// Mitsubishi GX Works2 project: 05.01Group17Final   PLC: FX3G

// global labels: Global1
VAR_GLOBAL
  Start_Day AT X007 : BOOL;
  Y_7 AT Y007 : BOOL;
  FillZilofKazefet AT X011 : BOOL;
  HelpLight AT M34 : BOOL;
  BlinkingLight AT M4 : BOOL;
  BlinkingTimer1 AT TC0 : BOOL;
  ConstantBlinking AT K5 : INT;
  TimerValue1 AT TS0 : BOOL;
  BlinkingLight2 AT M5 : BOOL;
  BlinkingTimer2 AT TC1 : BOOL;
  TimerValue2 AT TS1 : BOOL;
  BlinkingLightStop AT M5 : BOOL;
  StopBlinking AT TS4 : BOOL;
  Timer4 AT TC4 : BOOL;
  EndDay AT K30 : INT;
  BlinkingLightStop1 AT M6 : BOOL;
  CHOCOLATE AT D1111 : REAL;
  CREAM_STOCK AT D1118 : REAL;
  CHOCOLATE_STOCK AT D1121 : REAL;
  BISCUIT_STOCK AT D1124 : REAL;
END_VAR
VAR_GLOBAL CONSTANT
  C_300 : REAL := 300;
  C_260 : INT := 600;
  C_240 : REAL := 240;
  B_6 : REAL := 6;
END_VAR
VAR_GLOBAL
  VALID AT M2 : BOOL;
  CREAM AT D1100 : REAL;
  BISCUIT AT D1113 : REAL;
  X1_touch AT X001 : BOOL;
  X2_Cam AT X002 : BOOL;
  X5_error AT X005 : BOOL;
  System_on AT M0 : BOOL;
  x3_Sen_30 AT X003 : BOOL;
  X4_sen_15 AT X004 : BOOL;
  Spirk_system AT Y004 : BOOL;
  shut_Down AT X007 : BOOL;
  Start_sys AT X010 : BOOL;
  moveCream AT X011 : BOOL;
  sprinklingContainer AT D1127 : REAL;
END_VAR
VAR_GLOBAL CONSTANT
  nimus_300 : REAL := 300;
  minus_300 : REAL := 300;
  minus_6 : REAL := 6;
END_VAR
VAR_GLOBAL
  M_10 AT M10 : BOOL;
  TimerShinua AT TC10 : BOOL;
END_VAR
VAR_GLOBAL CONSTANT
  shinua : INT := 40;
END_VAR
VAR_GLOBAL
  shinuaFinished AT TS10 : BOOL;
  Y_0 AT Y000 : BOOL;
  Y_1 AT Y001 : BOOL;
  analogCheck AT X006 : BOOL;
  analogInput1 AT D8280 : INT;
  saveAnalog1 AT D1300 : INT;
END_VAR
VAR_GLOBAL CONSTANT
  lessThan : INT := 5;
  lessthan_10 : INT := 10;
  moreThan_6 : INT := 6;
END_VAR
VAR_GLOBAL
  less_10 : BOOL;
  Be0_5 AT M55 : BOOL;
  Be6_10 AT M56 : BOOL;
END_VAR
VAR_GLOBAL CONSTANT
  regularTzipuy : REAL := 120;
  doubleTzipuy : REAL := 240;
END_VAR
VAR_GLOBAL
  dipContainer AT D1132 : REAL;
  TimerDip AT TC8 : BOOL;
END_VAR
VAR_GLOBAL CONSTANT
  timer5 : INT := 50;
END_VAR
VAR_GLOBAL
  TS_8 AT TS8 : BOOL;
  Y_3 AT Y003 : BOOL;
  Gelem AT M80 : BOOL;
END_VAR
VAR_GLOBAL CONSTANT
  div400 : INT := 400;
END_VAR
VAR_GLOBAL
  M_100 AT M100 : BOOL;
  M_101 AT M101 : BOOL;
  ariza AT X000 : BOOL;
  countUnits AT CC0 : BOOL;
END_VAR
VAR_GLOBAL CONSTANT
  Equal_5 : REAL;
END_VAR
VAR_GLOBAL
  Y_2 AT Y002 : BOOL;
END_VAR
VAR_GLOBAL CONSTANT
  Mishtane : INT := 5;
END_VAR
VAR_GLOBAL
  CS_0 AT CS0 : BOOL;
  countUnits2 AT CC1 : BOOL;
END_VAR
VAR_GLOBAL CONSTANT
  until6 : INT := 6;
END_VAR
VAR_GLOBAL
  CS_1 AT CS1 : BOOL;
  rst_ziluf AT M60 : BOOL;
END_VAR
VAR_GLOBAL CONSTANT
  div10 : INT := 10;
END_VAR
VAR_GLOBAL
  Output_Analog1 AT D1150 : INT;
END_VAR
VAR_GLOBAL CONSTANT
  E_120 : INT := 120;
  E_240 : INT := 240;
  plus20 : INT := 20;
  limit : INT := 6;
  add_6 : INT := 6;
END_VAR
VAR_GLOBAL
  closeCount AT M77 : BOOL;
  M_EZER AT M99 : BOOL;
  M_reCheck AT M88 : BOOL;
END_VAR
VAR_GLOBAL CONSTANT
  last_6 : INT := 6;
END_VAR
VAR_GLOBAL
  count_last_6 AT CC12 : BOOL;
  EndOfDay AT CS12 : BOOL;
  analogOutput AT D8282 : INT;
END_VAR
VAR_GLOBAL CONSTANT
  mul40 : INT := 40;
END_VAR

// task Task_01 (event TRUE, interval 0, priority 31): POU_01

PROGRAM POU_01
VAR CONSTANT
  plus_one : INT := 1;
END_VAR
(* structured ladder/FBD written out as ST: instructions are called as NAME(EN, inputs, outputs); _pN, _eN, _tN stand for wires *)
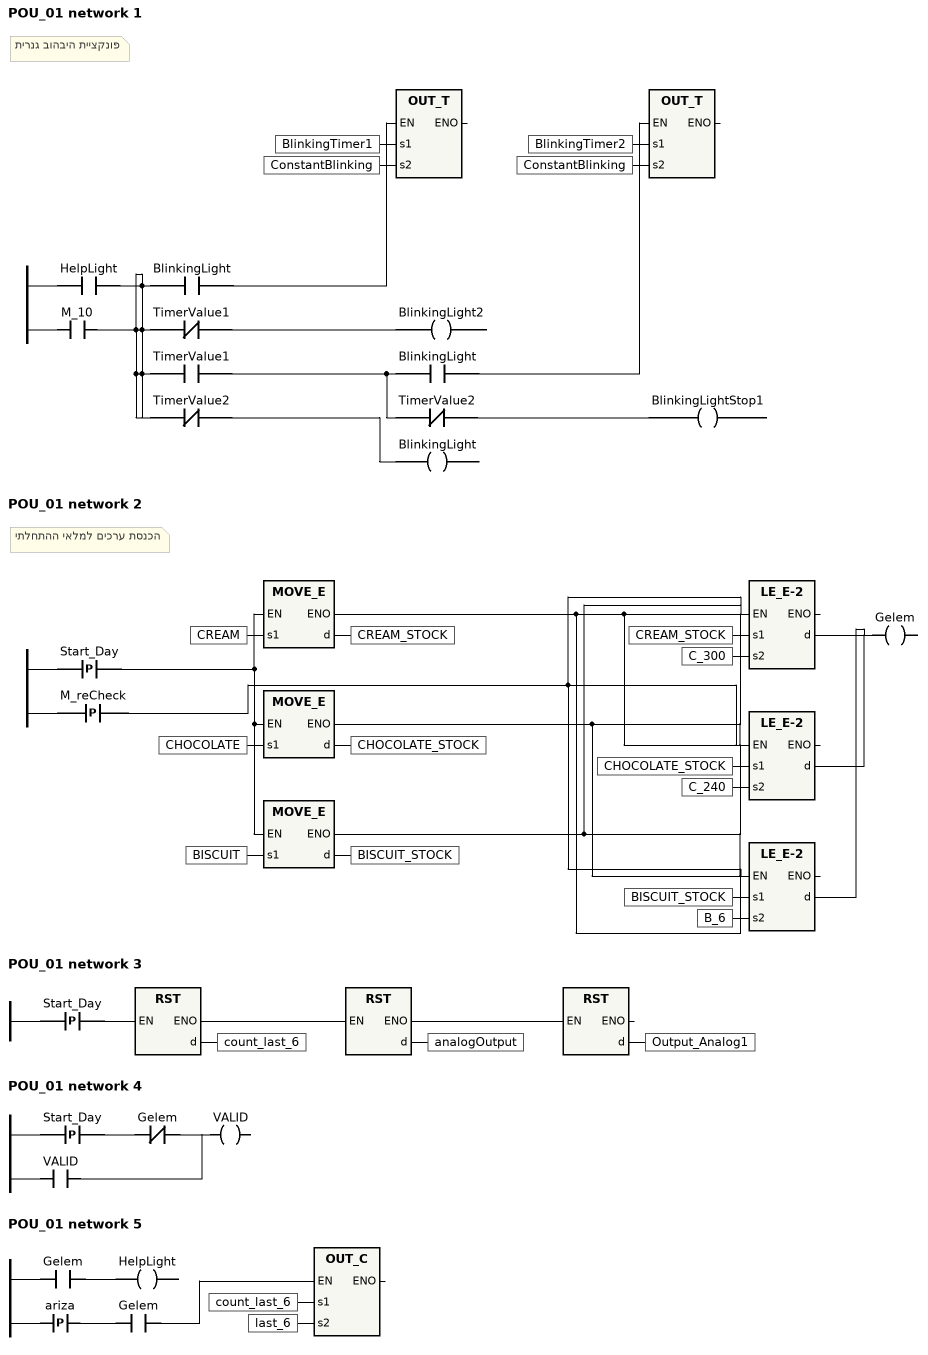
(* network 1 *)
(* פונקציית היבהוב גנרית *)
_p1 := HelpLight OR M_10;
OUT_T(_p1 AND BlinkingLight, BlinkingTimer1, ConstantBlinking);
BlinkingLight2 := _p1 AND NOT TimerValue1;
_p2 := _p1 AND TimerValue1;
OUT_T(_p2 AND BlinkingLight, BlinkingTimer2, ConstantBlinking);
BlinkingLightStop1 := _p2 AND NOT TimerValue2;
BlinkingLight := _p1 AND NOT TimerValue2;
(* network 2 *)
(* הכנסת ערכים למלאי ההתחלתי *)
_p1 := LDP(TRUE, Start_Day);
_e2 := MOVE_E(_p1, CREAM, CREAM_STOCK);
_e3 := MOVE_E(_p1, CHOCOLATE, CHOCOLATE_STOCK);
_e4 := MOVE_E(_p1, BISCUIT, BISCUIT_STOCK);
_p5 := _e2 OR _e3 OR _e4 OR LDP(TRUE, M_reCheck);
LE_E(_p5, CREAM_STOCK, C_300, _t6);
LE_E(_p5, CHOCOLATE_STOCK, C_240, _t7);
LE_E(_p5, BISCUIT_STOCK, B_6, _t8);
Gelem := _t6 OR _t7 OR _t8;
(* network 3 *)
_e1 := RST(LDP(TRUE, Start_Day), count_last_6);
_e2 := RST(_e1, analogOutput);
RST(_e2, Output_Analog1);
(* network 4 *)
VALID := (LDP(TRUE, Start_Day) AND NOT Gelem) OR VALID;
(* network 5 *)
HelpLight := Gelem;
OUT_C(LDP(TRUE, ariza) AND Gelem, count_last_6, last_6);
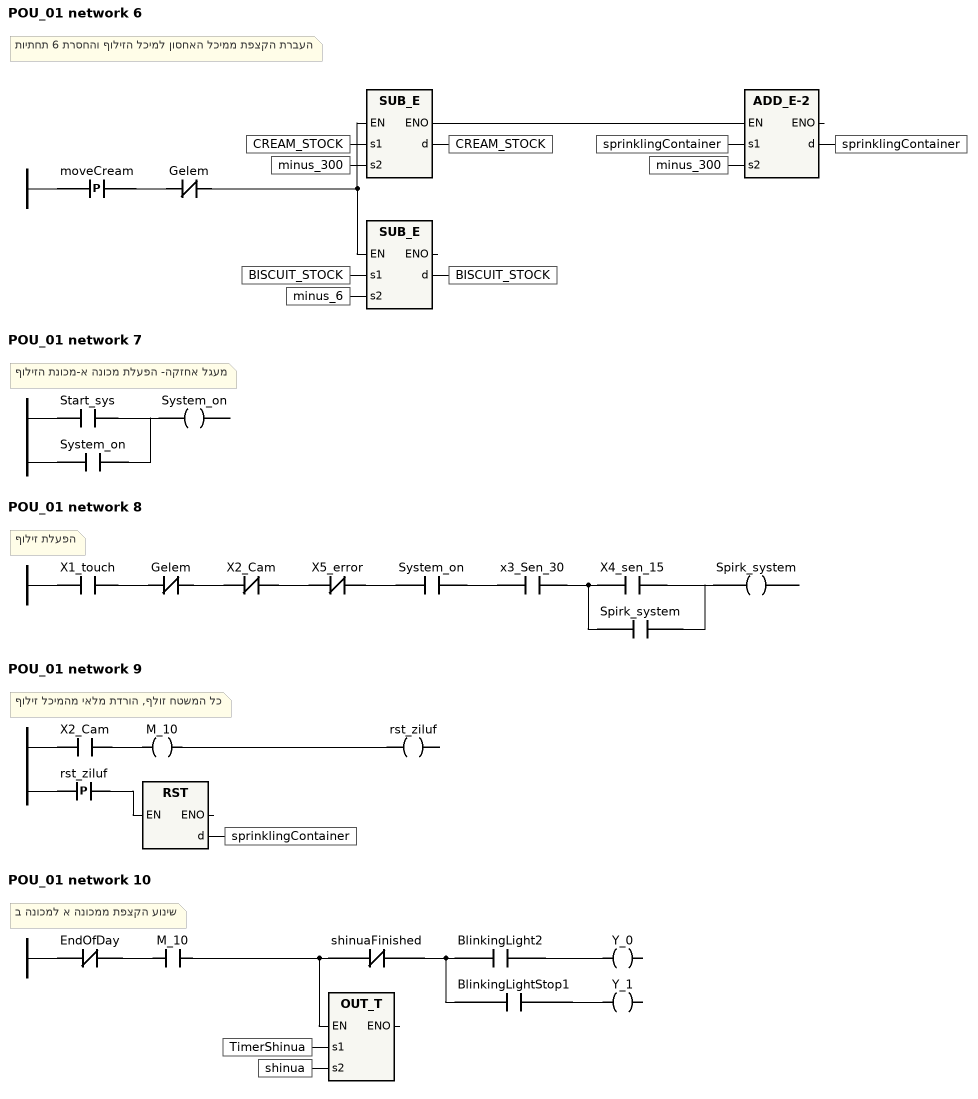
(* network 6 *)
(* העברת הקצפת ממיכל האחסון למיכל הזילוף והחסרת 6 תחתיות *)
_p1 := LDP(TRUE, moveCream) AND NOT Gelem;
_e2 := SUB_E(_p1, CREAM_STOCK, minus_300, CREAM_STOCK);
ADD_E(_e2, sprinklingContainer, minus_300, sprinklingContainer);
SUB_E(_p1, BISCUIT_STOCK, minus_6, BISCUIT_STOCK);
(* network 7 *)
(* מעגל אחזקה- הפעלת מכונה א-מכונת הזילוף *)
System_on := Start_sys OR System_on;
(* network 8 *)
(* הפעלת זילוף *)
_p1 := X1_touch AND NOT Gelem AND NOT X2_Cam AND NOT X5_error AND System_on AND x3_Sen_30;
Spirk_system := (_p1 AND X4_sen_15) OR (_p1 AND Spirk_system);
(* network 9 *)
(* כל המשטח זולף, הורדת מלאי מהמיכל זילוף *)
M_10 := X2_Cam;
rst_ziluf := X2_Cam;
RST(LDP(TRUE, rst_ziluf), sprinklingContainer);
(* network 10 *)
(* שינוע הקצפת ממכונה א למכונה ב *)
_p1 := NOT EndOfDay AND M_10;
_p2 := _p1 AND NOT shinuaFinished;
Y_0 := _p2 AND BlinkingLight2;
OUT_T(_p1, TimerShinua, shinua);
Y_1 := _p2 AND BlinkingLightStop1;
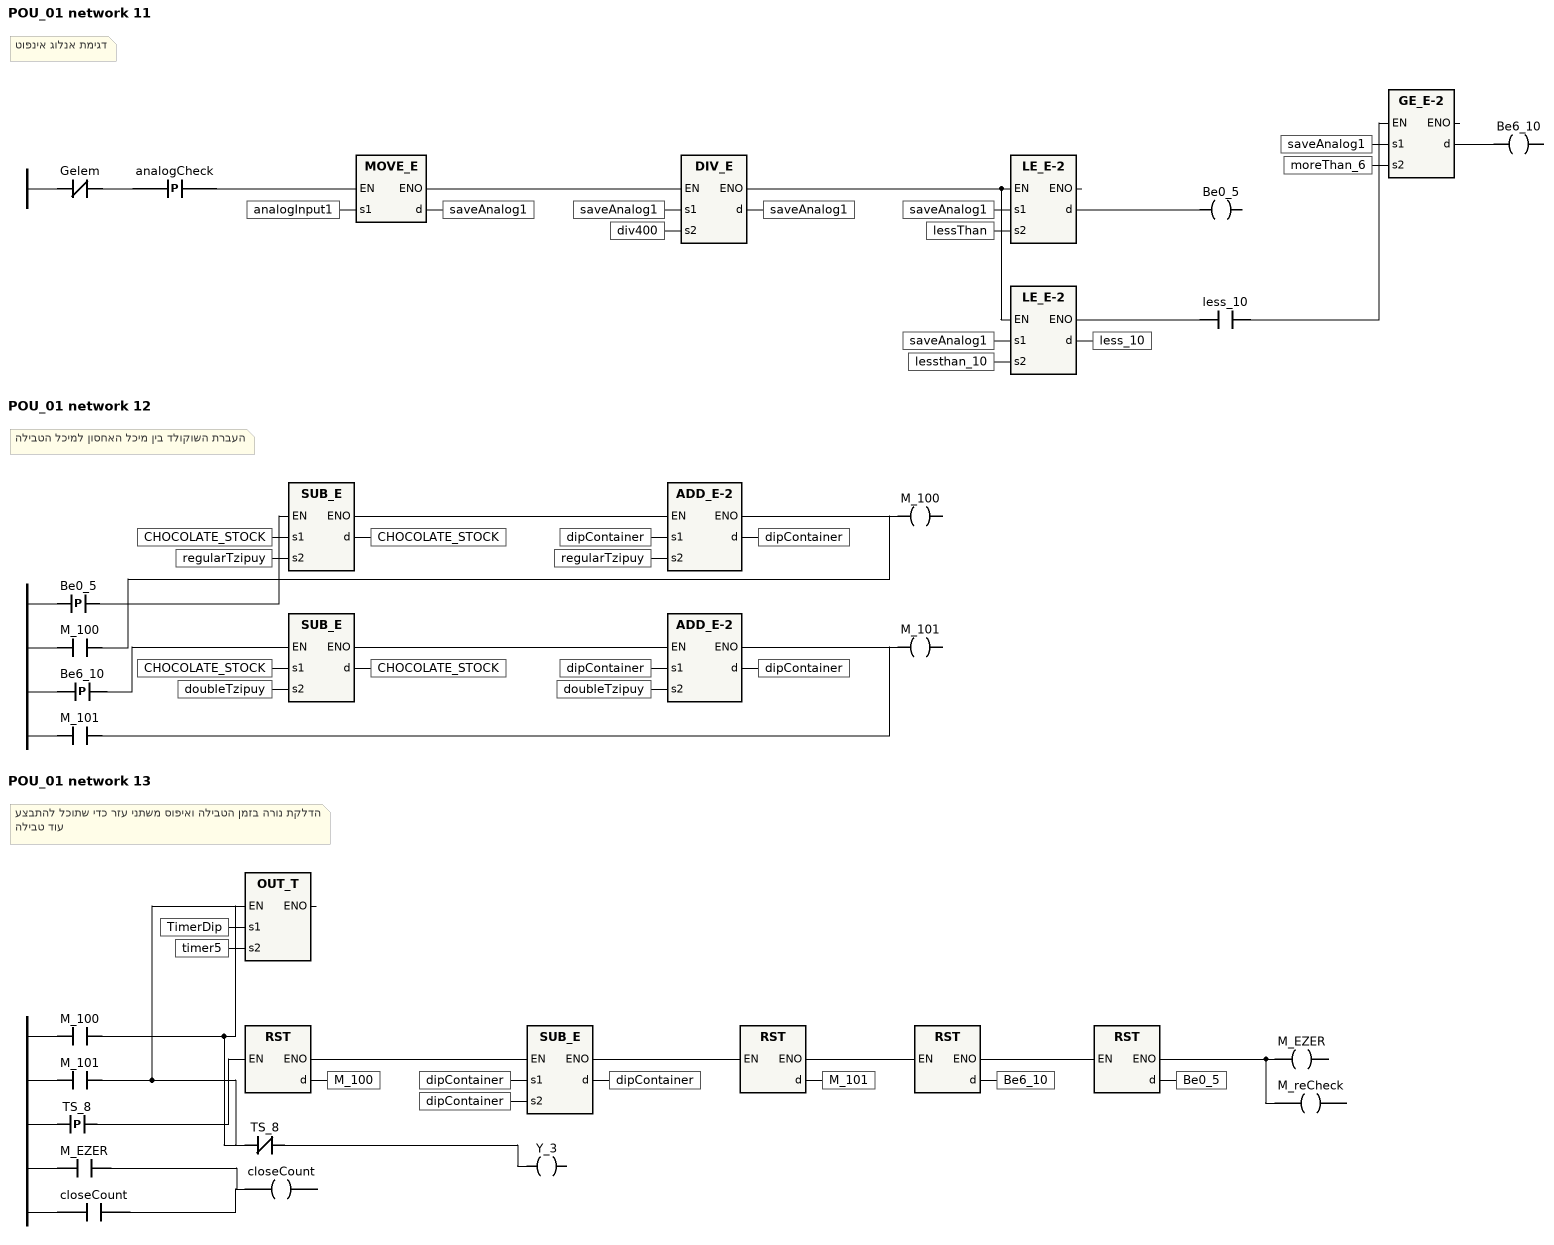
(* network 11 *)
(* דגימת אנלוג אינפוט *)
_e1 := MOVE_E(NOT Gelem AND LDP(TRUE, analogCheck), analogInput1, saveAnalog1);
_e2 := DIV_E(_e1, saveAnalog1, div400, saveAnalog1);
LE_E(_e2, saveAnalog1, lessThan, _t3);
Be0_5 := _t3;
_e4 := LE_E(_e2, saveAnalog1, lessthan_10, less_10);
GE_E(_e4 AND less_10, saveAnalog1, moreThan_6, _t5);
Be6_10 := _t5;
(* network 12 *)
(* העברת השוקולד בין מיכל האחסון למיכל הטבילה *)
_e1 := SUB_E(LDP(TRUE, Be0_5), CHOCOLATE_STOCK, regularTzipuy, CHOCOLATE_STOCK);
_e2 := ADD_E(_e1, dipContainer, regularTzipuy, dipContainer);
M_100 := _e2 OR M_100;
_e3 := SUB_E(LDP(TRUE, Be6_10), CHOCOLATE_STOCK, doubleTzipuy, CHOCOLATE_STOCK);
_e4 := ADD_E(_e3, dipContainer, doubleTzipuy, dipContainer);
M_101 := _e4 OR M_101;
(* network 13 *)
(* הדלקת נורה בזמן הטבילה ואיפוס משתני עזר כדי שתוכל להתבצע עוד טבילה *)
_p1 := M_100 OR M_101;
Y_3 := _p1 AND NOT TS_8;
OUT_T(_p1, TimerDip, timer5);
_e2 := RST(LDP(TRUE, TS_8), M_100);
_e3 := SUB_E(_e2, dipContainer, dipContainer, dipContainer);
_e4 := RST(_e3, M_101);
_e5 := RST(_e4, Be6_10);
_e6 := RST(_e5, Be0_5);
M_EZER := _e6;
M_reCheck := _e6;
closeCount := M_EZER OR closeCount;
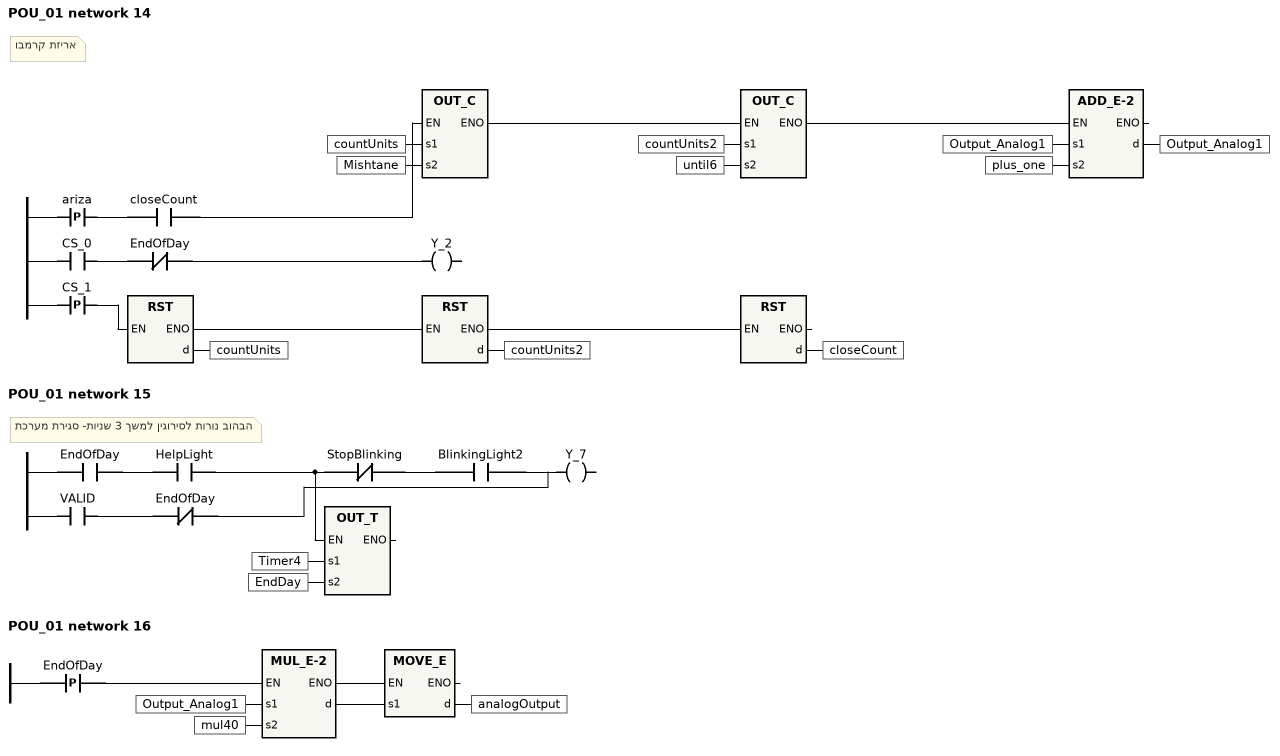
(* network 14 *)
(* אריזת קרמבו *)
_e1 := OUT_C(LDP(TRUE, ariza) AND closeCount, countUnits, Mishtane);
_e2 := OUT_C(_e1, countUnits2, until6);
ADD_E(_e2, Output_Analog1, plus_one, Output_Analog1);
Y_2 := CS_0 AND NOT EndOfDay;
_e3 := RST(LDP(TRUE, CS_1), countUnits);
_e4 := RST(_e3, countUnits2);
RST(_e4, closeCount);
(* network 15 *)
(* הבהוב נורות לסירוגין למשך 3 שניות- סגירת מערכת *)
_p1 := EndOfDay AND HelpLight;
Y_7 := (_p1 AND NOT StopBlinking AND BlinkingLight2) OR (VALID AND NOT EndOfDay);
OUT_T(_p1, Timer4, EndDay);
(* network 16 *)
_e2 := MUL_E(LDP(TRUE, EndOfDay), Output_Analog1, mul40, _t1);
MOVE_E(_e2, _t1, analogOutput);
END_PROGRAM
